// Mitsubishi GX Developer project: 20170103   PLC: FX1N

PROGRAM MAIN
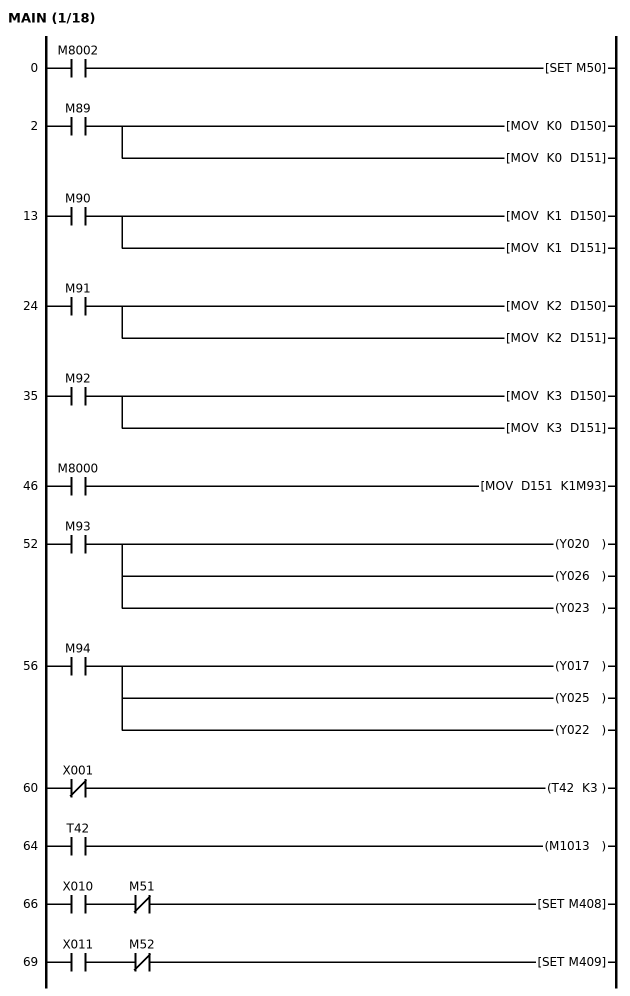
0     LD      M8002
      SET     M50
2     LD      M89
      MOV     K0 D150
      MOV     K0 D151
13    LD      M90
      MOV     K1 D150
      MOV     K1 D151
24    LD      M91
      MOV     K2 D150
      MOV     K2 D151
35    LD      M92
      MOV     K3 D150
      MOV     K3 D151
46    LD      M8000
      MOV     D151 K1M93
52    LD      M93
      OUT     Y020
      OUT     Y026
      OUT     Y023
56    LD      M94
      OUT     Y017
      OUT     Y025
      OUT     Y022
60    LDI     X001
      OUT     T42 K3
64    LD      T42
      OUT     M1013
66    LD      X010
      ANI     M51
      SET     M408
69    LD      X011
      ANI     M52
      SET     M409
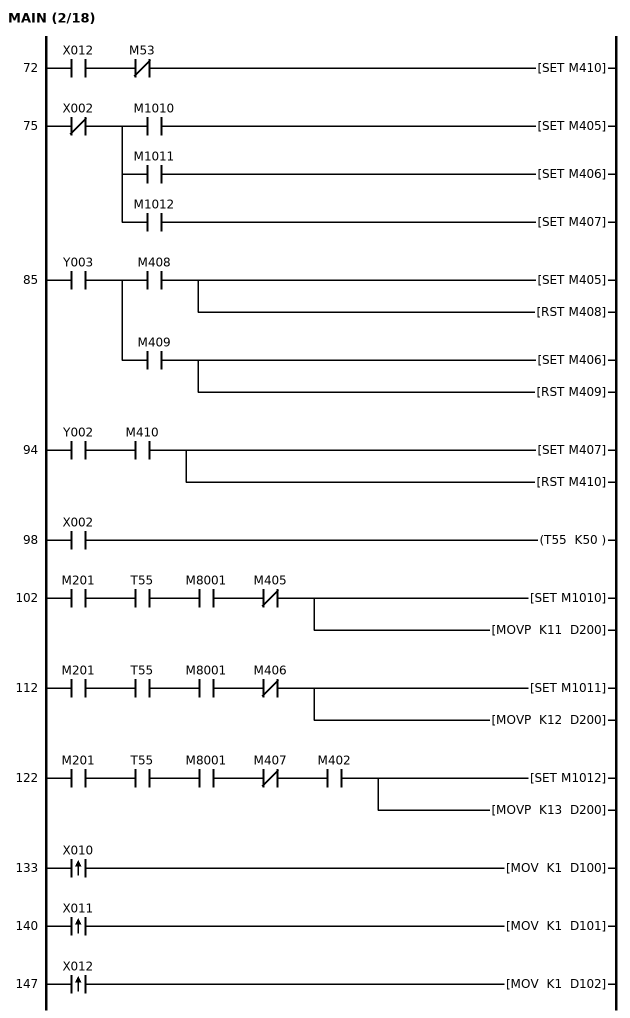
72    LD      X012
      ANI     M53
      SET     M410
75    LDI     X002
      MPS
      AND     M1010
      SET     M405
      MRD
      AND     M1011
      SET     M406
      MPP
      AND     M1012
      SET     M407
85    LD      Y003
      MPS
      AND     M408
      SET     M405
      RST     M408
      MPP
      AND     M409
      SET     M406
      RST     M409
94    LD      Y002
      AND     M410
      SET     M407
      RST     M410
98    LD      X002
      OUT     T55 K50
102   LD      M201
      AND     T55
      AND     M8001
      ANI     M405
      SET     M1010
      MOVP    K11 D200
112   LD      M201
      AND     T55
      AND     M8001
      ANI     M406
      SET     M1011
      MOVP    K12 D200
122   LD      M201
      AND     T55
      AND     M8001
      ANI     M407
      AND     M402
      SET     M1012
      MOVP    K13 D200
133   LDP     X010
      MOV     K1 D100
140   LDP     X011
      MOV     K1 D101
147   LDP     X012
      MOV     K1 D102
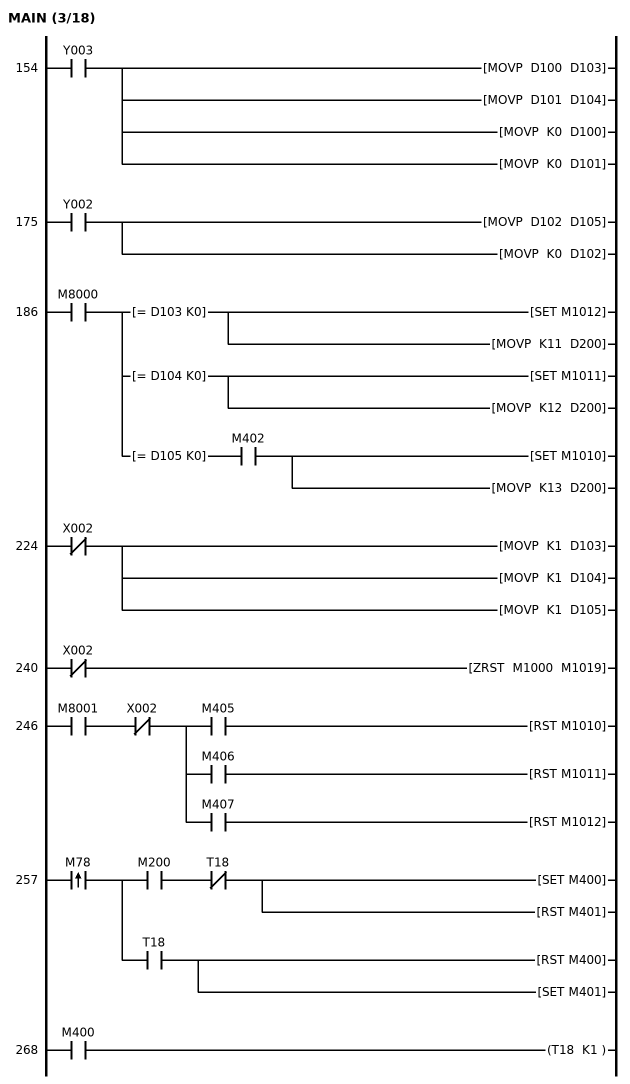
154   LD      Y003
      MOVP    D100 D103
      MOVP    D101 D104
      MOVP    K0 D100
      MOVP    K0 D101
175   LD      Y002
      MOVP    D102 D105
      MOVP    K0 D102
186   LD      M8000
      MPS
      AND=    D103 K0
      SET     M1012
      MOVP    K11 D200
      MRD
      AND=    D104 K0
      SET     M1011
      MOVP    K12 D200
      MPP
      AND=    D105 K0
      AND     M402
      SET     M1010
      MOVP    K13 D200
224   LDI     X002
      MOVP    K1 D103
      MOVP    K1 D104
      MOVP    K1 D105
240   LDI     X002
      ZRST    M1000 M1019
246   LD      M8001
      ANI     X002
      MPS
      AND     M405
      RST     M1010
      MRD
      AND     M406
      RST     M1011
      MPP
      AND     M407
      RST     M1012
257   LDP     M78
      MPS
      AND     M200
      ANI     T18
      SET     M400
      RST     M401
      MPP
      AND     T18
      RST     M400
      SET     M401
268   LD      M400
      OUT     T18 K1
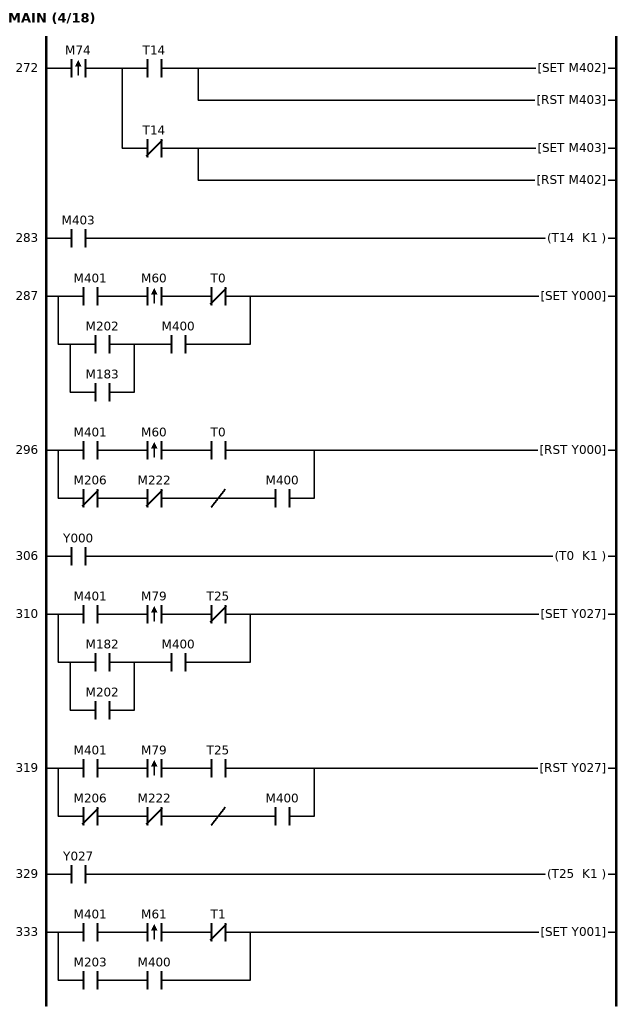
272   LDP     M74
      MPS
      AND     T14
      SET     M402
      RST     M403
      MPP
      ANI     T14
      SET     M403
      RST     M402
283   LD      M403
      OUT     T14 K1
287   LD      M401
      ANDP    M60
      ANI     T0
      LD      M202
      OR      M183
      AND     M400
      ORB
      SET     Y000
296   LD      M401
      ANDP    M60
      AND     T0
      LDI     M206
      ANI     M222
      INV
      AND     M400
      ORB
      RST     Y000
306   LD      Y000
      OUT     T0 K1
310   LD      M401
      ANDP    M79
      ANI     T25
      LD      M182
      OR      M202
      AND     M400
      ORB
      SET     Y027
319   LD      M401
      ANDP    M79
      AND     T25
      LDI     M206
      ANI     M222
      INV
      AND     M400
      ORB
      RST     Y027
329   LD      Y027
      OUT     T25 K1
333   LD      M401
      ANDP    M61
      ANI     T1
      LD      M203
      AND     M400
      ORB
      SET     Y001
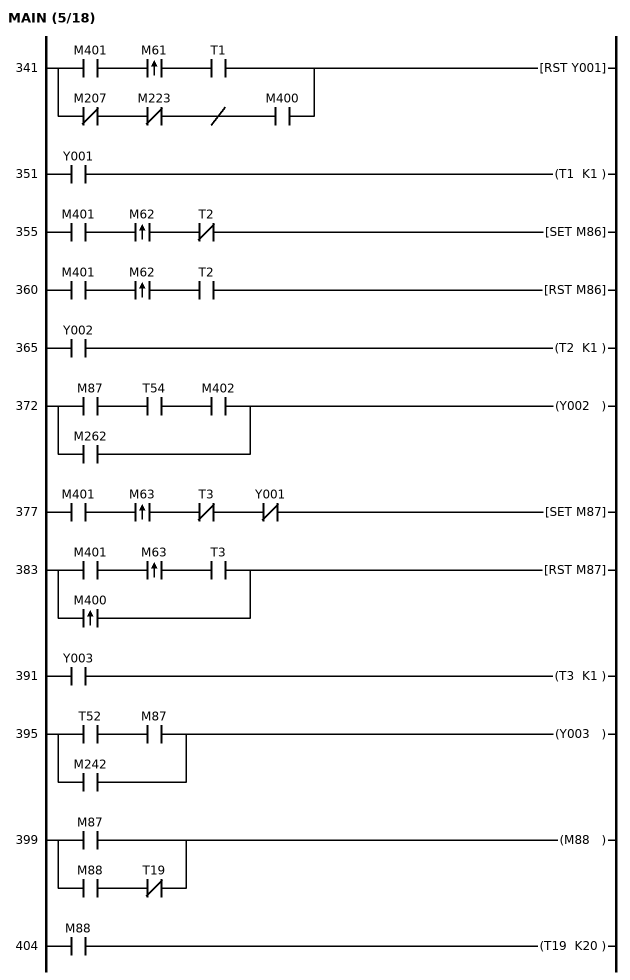
341   LD      M401
      ANDP    M61
      AND     T1
      LDI     M207
      ANI     M223
      INV
      AND     M400
      ORB
      RST     Y001
351   LD      Y001
      OUT     T1 K1
355   LD      M401
      ANDP    M62
      ANI     T2
      SET     M86
360   LD      M401
      ANDP    M62
      AND     T2
      RST     M86
365   LD      Y002
      OUT     T2 K1
372   LD      M87
      AND     T54
      AND     M402
      OR      M262
      OUT     Y002
377   LD      M401
      ANDP    M63
      ANI     T3
      ANI     Y001
      SET     M87
383   LD      M401
      ANDP    M63
      AND     T3
      ORP     M400
      RST     M87
391   LD      Y003
      OUT     T3 K1
395   LD      T52
      AND     M87
      OR      M242
      OUT     Y003
399   LD      M87
      LD      M88
      ANI     T19
      ORB
      OUT     M88
404   LD      M88
      OUT     T19 K20
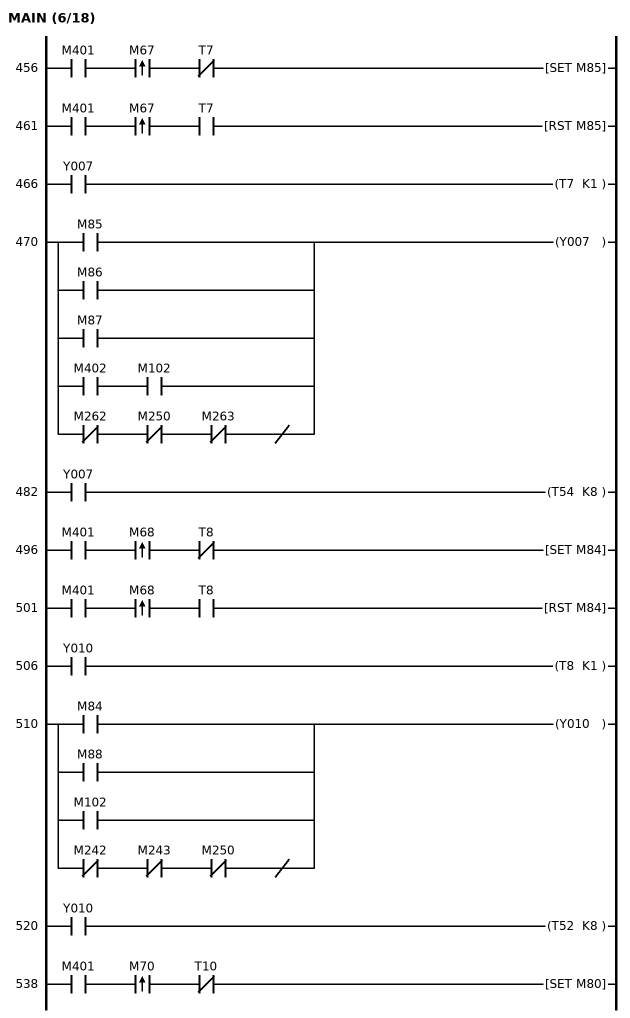
456   LD      M401
      ANDP    M67
      ANI     T7
      SET     M85
461   LD      M401
      ANDP    M67
      AND     T7
      RST     M85
466   LD      Y007
      OUT     T7 K1
470   LD      M85
      OR      M86
      OR      M87
      LD      M402
      AND     M102
      ORB
      LDI     M262
      ANI     M250
      ANI     M263
      INV
      ORB
      OUT     Y007
482   LD      Y007
      OUT     T54 K8
496   LD      M401
      ANDP    M68
      ANI     T8
      SET     M84
501   LD      M401
      ANDP    M68
      AND     T8
      RST     M84
506   LD      Y010
      OUT     T8 K1
510   LD      M84
      OR      M88
      OR      M102
      LDI     M242
      ANI     M243
      ANI     M250
      INV
      ORB
      OUT     Y010
520   LD      Y010
      OUT     T52 K8
538   LD      M401
      ANDP    M70
      ANI     T10
      SET     M80
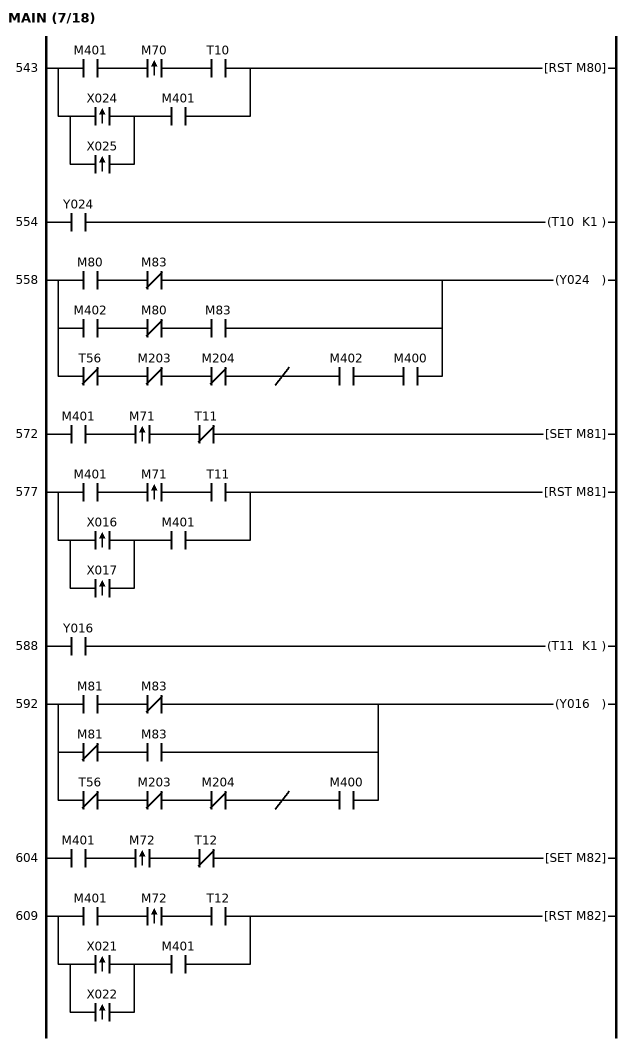
543   LD      M401
      ANDP    M70
      AND     T10
      LDP     X024
      ORP     X025
      AND     M401
      ORB
      RST     M80
554   LD      Y024
      OUT     T10 K1
558   LD      M80
      ANI     M83
      LD      M402
      ANI     M80
      AND     M83
      ORB
      LDI     T56
      ANI     M203
      ANI     M204
      INV
      AND     M402
      AND     M400
      ORB
      OUT     Y024
572   LD      M401
      ANDP    M71
      ANI     T11
      SET     M81
577   LD      M401
      ANDP    M71
      AND     T11
      LDP     X016
      ORP     X017
      AND     M401
      ORB
      RST     M81
588   LD      Y016
      OUT     T11 K1
592   LD      M81
      ANI     M83
      LDI     M81
      AND     M83
      ORB
      LDI     T56
      ANI     M203
      ANI     M204
      INV
      AND     M400
      ORB
      OUT     Y016
604   LD      M401
      ANDP    M72
      ANI     T12
      SET     M82
609   LD      M401
      ANDP    M72
      AND     T12
      LDP     X021
      ORP     X022
      AND     M401
      ORB
      RST     M82
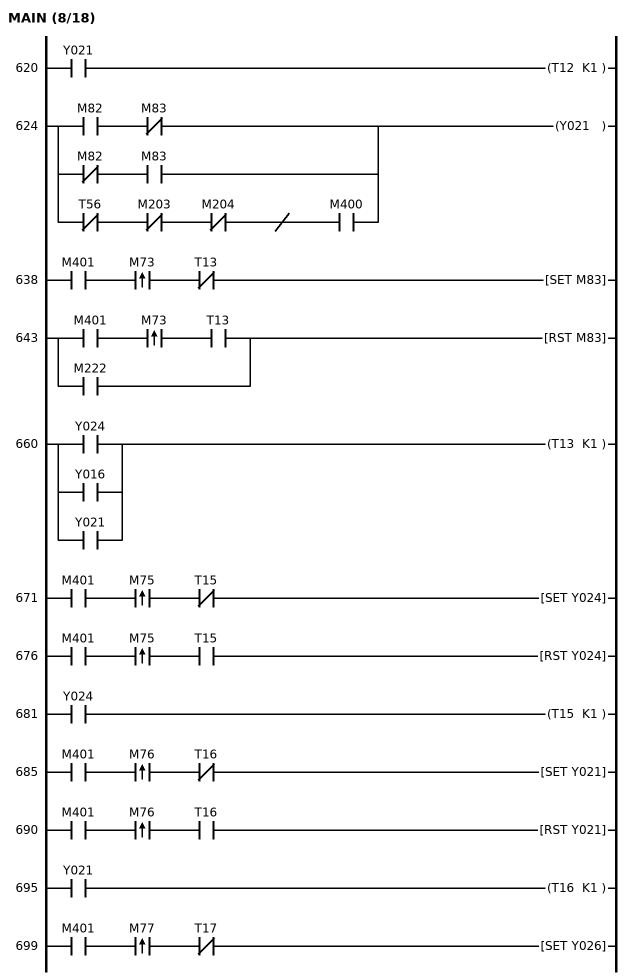
620   LD      Y021
      OUT     T12 K1
624   LD      M82
      ANI     M83
      LDI     M82
      AND     M83
      ORB
      LDI     T56
      ANI     M203
      ANI     M204
      INV
      AND     M400
      ORB
      OUT     Y021
638   LD      M401
      ANDP    M73
      ANI     T13
      SET     M83
643   LD      M401
      ANDP    M73
      AND     T13
      OR      M222
      RST     M83
660   LD      Y024
      OR      Y016
      OR      Y021
      OUT     T13 K1
671   LD      M401
      ANDP    M75
      ANI     T15
      SET     Y024
676   LD      M401
      ANDP    M75
      AND     T15
      RST     Y024
681   LD      Y024
      OUT     T15 K1
685   LD      M401
      ANDP    M76
      ANI     T16
      SET     Y021
690   LD      M401
      ANDP    M76
      AND     T16
      RST     Y021
695   LD      Y021
      OUT     T16 K1
699   LD      M401
      ANDP    M77
      ANI     T17
      SET     Y026
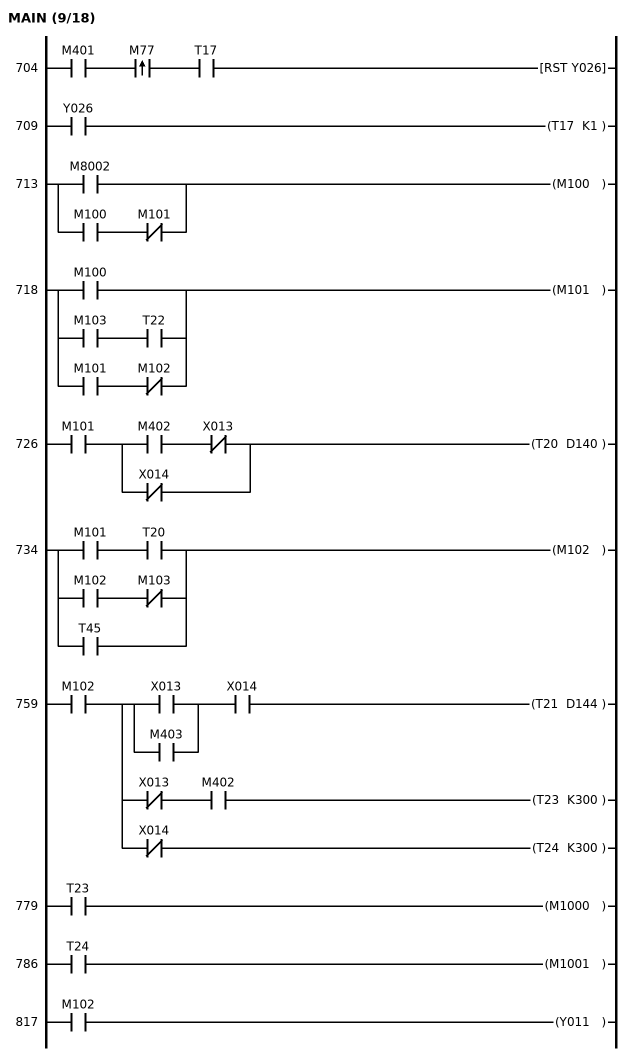
704   LD      M401
      ANDP    M77
      AND     T17
      RST     Y026
709   LD      Y026
      OUT     T17 K1
713   LD      M8002
      LD      M100
      ANI     M101
      ORB
      OUT     M100
718   LD      M100
      LD      M103
      AND     T22
      ORB
      LD      M101
      ANI     M102
      ORB
      OUT     M101
726   LD      M101
      LD      M402
      ANI     X013
      ORI     X014
      ANB
      OUT     T20 D140
734   LD      M101
      AND     T20
      LD      M102
      ANI     M103
      ORB
      OR      T45
      OUT     M102
759   LD      M102
      MPS
      LD      X013
      OR      M403
      ANB
      AND     X014
      OUT     T21 D144
      MRD
      ANI     X013
      AND     M402
      OUT     T23 K300
      MPP
      ANI     X014
      OUT     T24 K300
779   LD      T23
      OUT     M1000
786   LD      T24
      OUT     M1001
817   LD      M102
      OUT     Y011
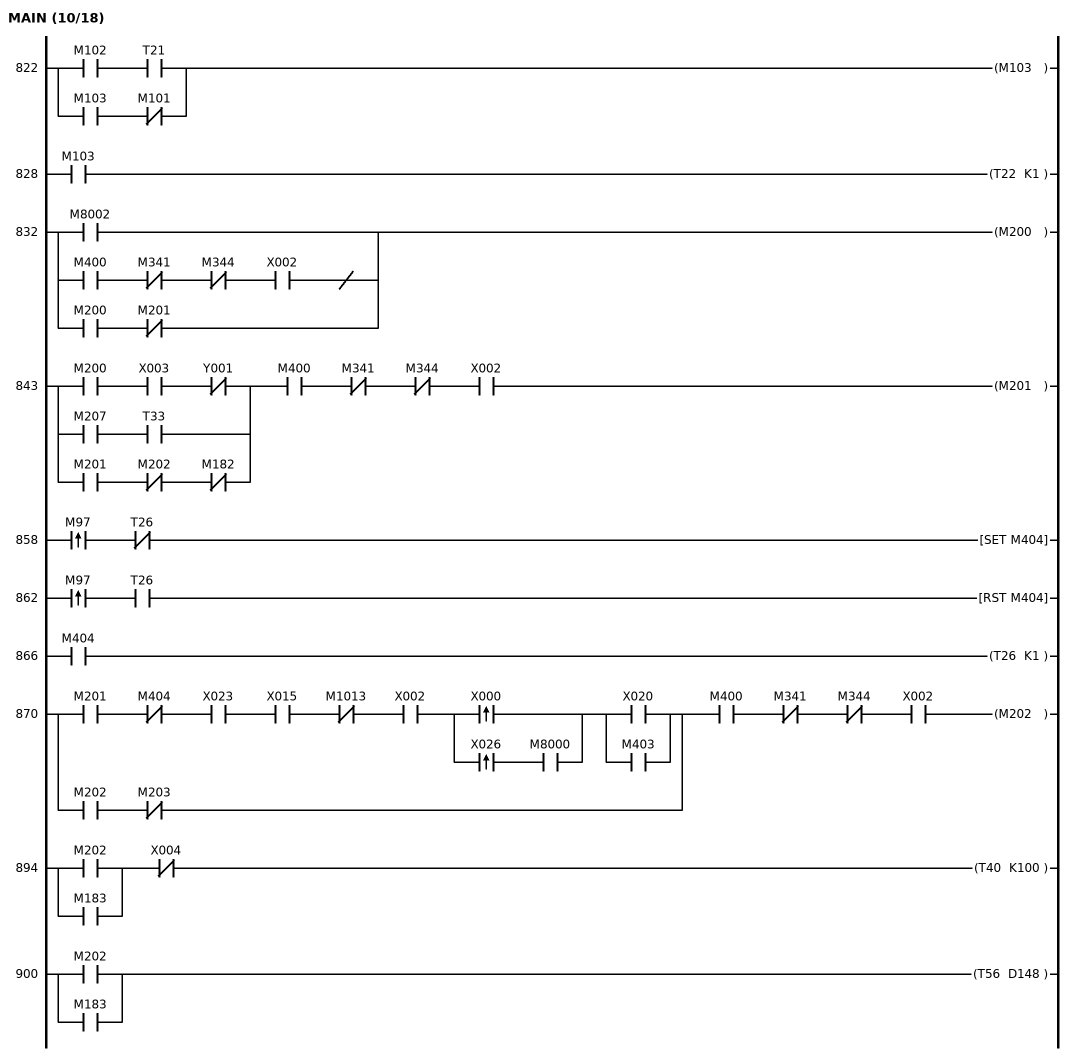
822   LD      M102
      AND     T21
      LD      M103
      ANI     M101
      ORB
      OUT     M103
828   LD      M103
      OUT     T22 K1
832   LD      M8002
      LD      M400
      ANI     M341
      ANI     M344
      AND     X002
      INV
      ORB
      LD      M200
      ANI     M201
      ORB
      OUT     M200
843   LD      M200
      AND     X003
      ANI     Y001
      LD      M207
      AND     T33
      ORB
      LD      M201
      ANI     M202
      ANI     M182
      ORB
      AND     M400
      ANI     M341
      ANI     M344
      AND     X002
      OUT     M201
858   LDP     M97
      ANI     T26
      SET     M404
862   LDP     M97
      AND     T26
      RST     M404
866   LD      M404
      OUT     T26 K1
870   LD      M201
      ANI     M404
      AND     X023
      AND     X015
      ANI     M1013
      AND     X002
      LDP     X000
      LDP     X026
      AND     M8000
      ORB
      ANB
      LD      X020
      OR      M403
      ANB
      LD      M202
      ANI     M203
      ORB
      AND     M400
      ANI     M341
      ANI     M344
      AND     X002
      OUT     M202
894   LD      M202
      OR      M183
      ANI     X004
      OUT     T40 K100
900   LD      M202
      OR      M183
      OUT     T56 D148
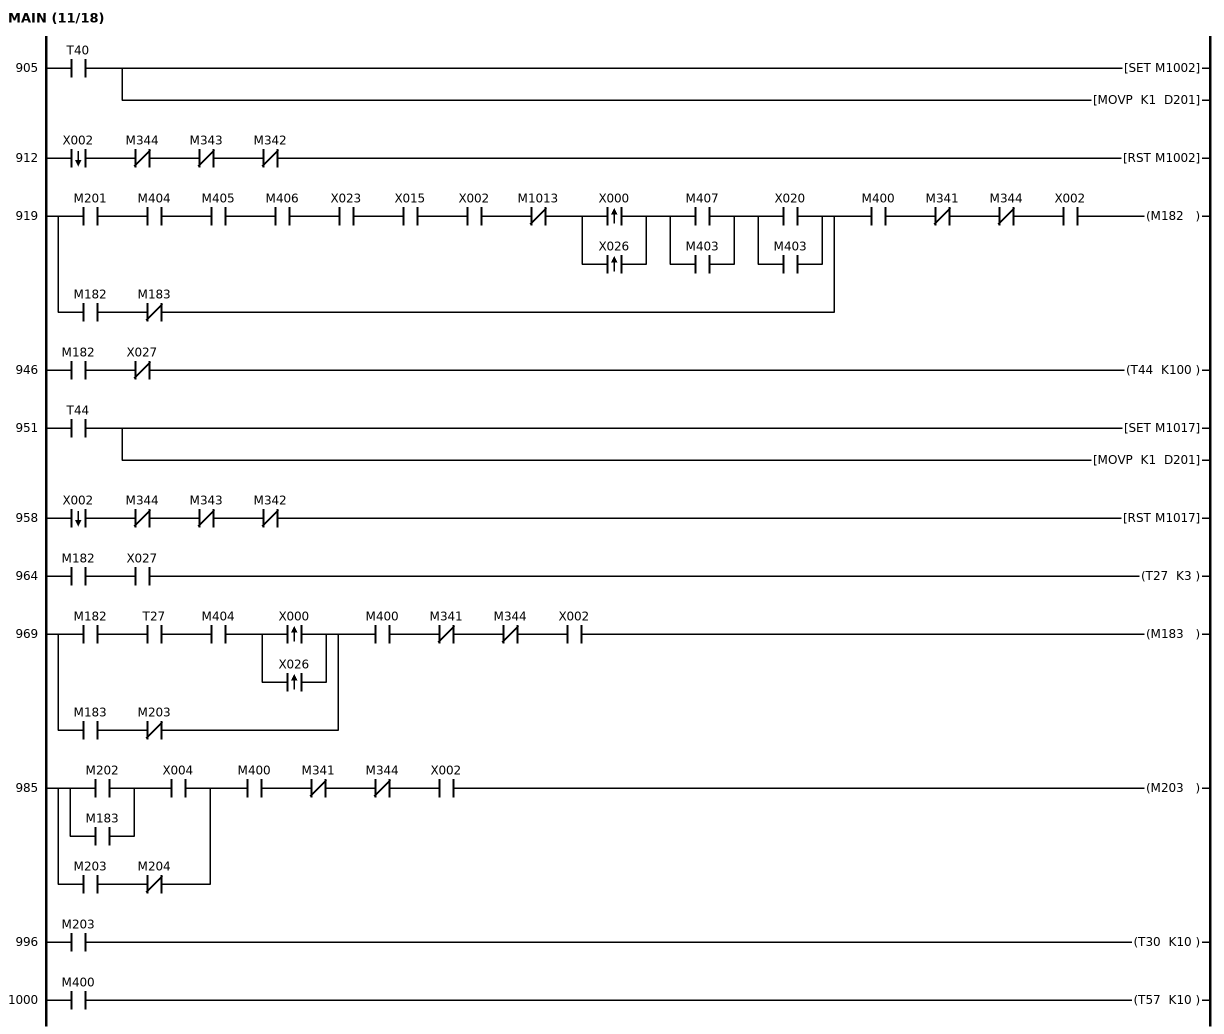
905   LD      T40
      SET     M1002
      MOVP    K1 D201
912   LDF     X002
      ANI     M344
      ANI     M343
      ANI     M342
      RST     M1002
919   LD      M201
      AND     M404
      AND     M405
      AND     M406
      AND     X023
      AND     X015
      AND     X002
      ANI     M1013
      LDP     X000
      ORP     X026
      ANB
      LD      M407
      OR      M403
      ANB
      LD      X020
      OR      M403
      ANB
      LD      M182
      ANI     M183
      ORB
      AND     M400
      ANI     M341
      ANI     M344
      AND     X002
      OUT     M182
946   LD      M182
      ANI     X027
      OUT     T44 K100
951   LD      T44
      SET     M1017
      MOVP    K1 D201
958   LDF     X002
      ANI     M344
      ANI     M343
      ANI     M342
      RST     M1017
964   LD      M182
      AND     X027
      OUT     T27 K3
969   LD      M182
      AND     T27
      AND     M404
      LDP     X000
      ORP     X026
      ANB
      LD      M183
      ANI     M203
      ORB
      AND     M400
      ANI     M341
      ANI     M344
      AND     X002
      OUT     M183
985   LD      M202
      OR      M183
      AND     X004
      LD      M203
      ANI     M204
      ORB
      AND     M400
      ANI     M341
      ANI     M344
      AND     X002
      OUT     M203
996   LD      M203
      OUT     T30 K10
1000  LD      M400
      OUT     T57 K10
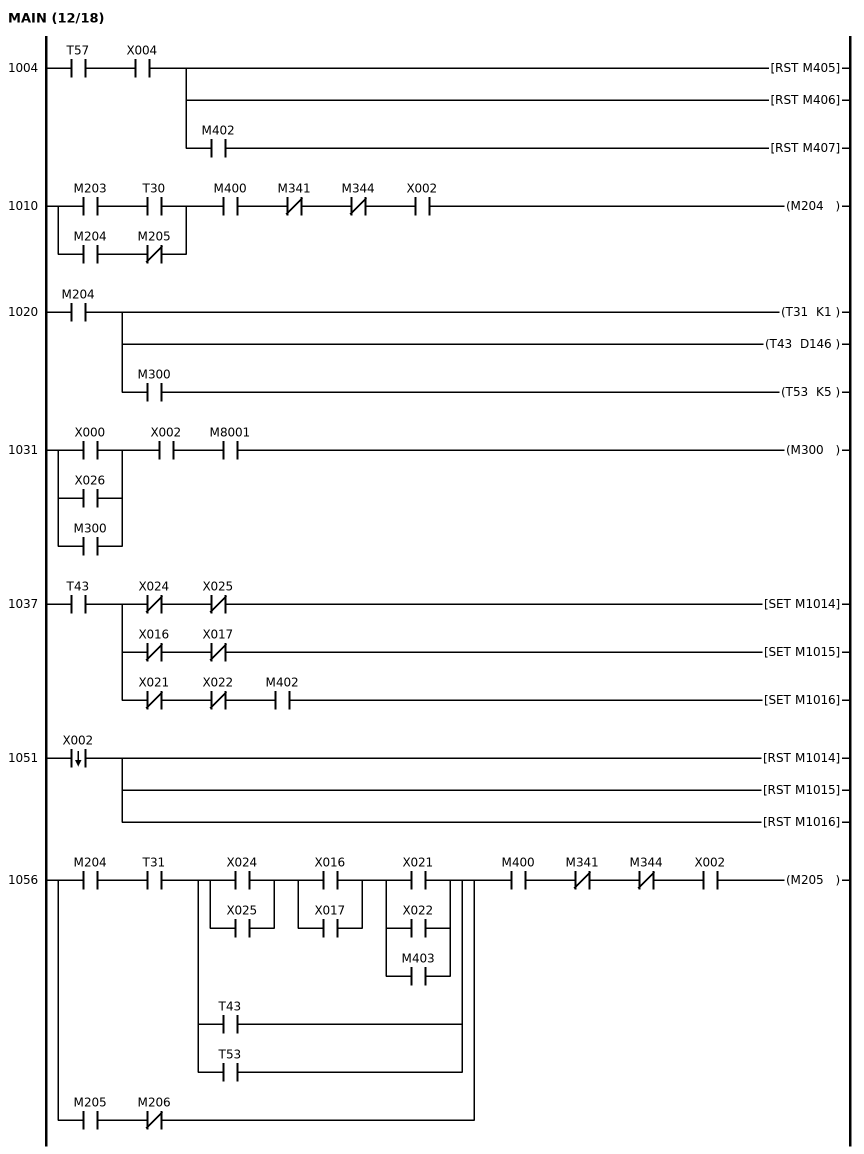
1004  LD      T57
      AND     X004
      RST     M405
      RST     M406
      AND     M402
      RST     M407
1010  LD      M203
      AND     T30
      LD      M204
      ANI     M205
      ORB
      AND     M400
      ANI     M341
      ANI     M344
      AND     X002
      OUT     M204
1020  LD      M204
      OUT     T31 K1
      OUT     T43 D146
      AND     M300
      OUT     T53 K5
1031  LD      X000
      OR      X026
      OR      M300
      AND     X002
      AND     M8001
      OUT     M300
1037  LD      T43
      MPS
      ANI     X024
      ANI     X025
      SET     M1014
      MRD
      ANI     X016
      ANI     X017
      SET     M1015
      MPP
      ANI     X021
      ANI     X022
      AND     M402
      SET     M1016
1051  LDF     X002
      RST     M1014
      RST     M1015
      RST     M1016
1056  LD      M204
      AND     T31
      LD      X024
      OR      X025
      LD      X016
      OR      X017
      ANB
      LD      X021
      OR      X022
      OR      M403
      ANB
      OR      T43
      OR      T53
      ANB
      LD      M205
      ANI     M206
      ORB
      AND     M400
      ANI     M341
      ANI     M344
      AND     X002
      OUT     M205
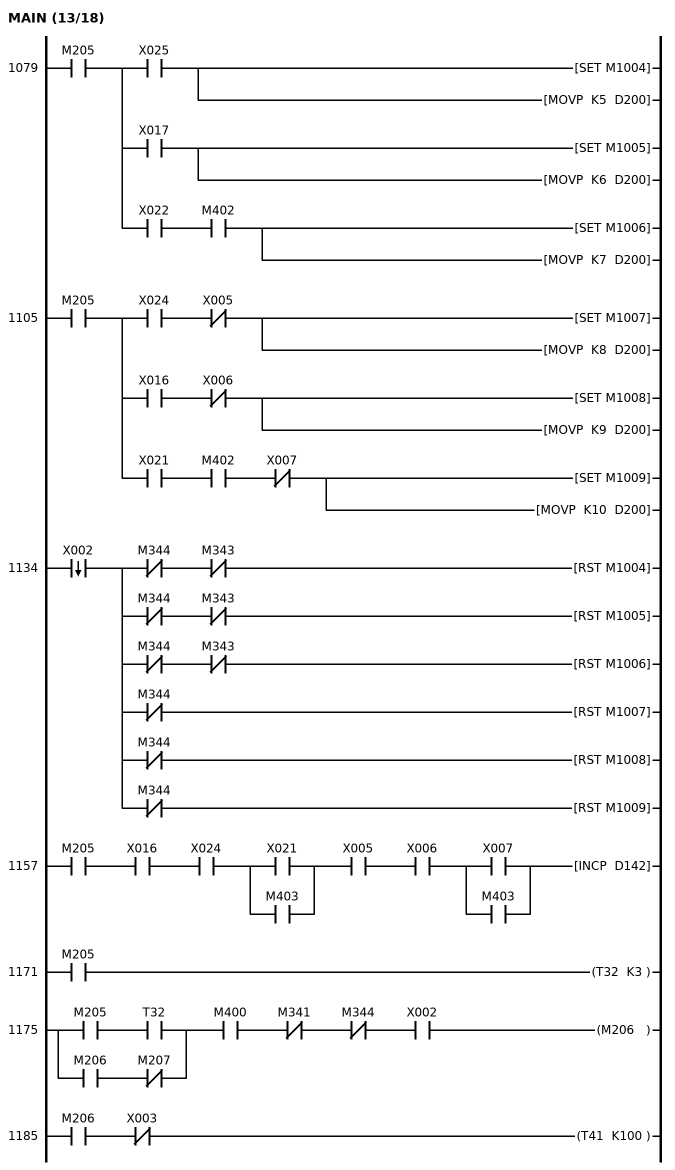
1079  LD      M205
      MPS
      AND     X025
      SET     M1004
      MOVP    K5 D200
      MRD
      AND     X017
      SET     M1005
      MOVP    K6 D200
      MPP
      AND     X022
      AND     M402
      SET     M1006
      MOVP    K7 D200
1105  LD      M205
      MPS
      AND     X024
      ANI     X005
      SET     M1007
      MOVP    K8 D200
      MRD
      AND     X016
      ANI     X006
      SET     M1008
      MOVP    K9 D200
      MPP
      AND     X021
      AND     M402
      ANI     X007
      SET     M1009
      MOVP    K10 D200
1134  LDF     X002
      MPS
      ANI     M344
      ANI     M343
      RST     M1004
      MRD
      ANI     M344
      ANI     M343
      RST     M1005
      MRD
      ANI     M344
      ANI     M343
      RST     M1006
      MRD
      ANI     M344
      RST     M1007
      MRD
      ANI     M344
      RST     M1008
      MPP
      ANI     M344
      RST     M1009
1157  LD      M205
      AND     X016
      AND     X024
      LD      X021
      OR      M403
      ANB
      AND     X005
      AND     X006
      LD      X007
      OR      M403
      ANB
      INCP    D142
1171  LD      M205
      OUT     T32 K3
1175  LD      M205
      AND     T32
      LD      M206
      ANI     M207
      ORB
      AND     M400
      ANI     M341
      ANI     M344
      AND     X002
      OUT     M206
1185  LD      M206
      ANI     X003
      OUT     T41 K100
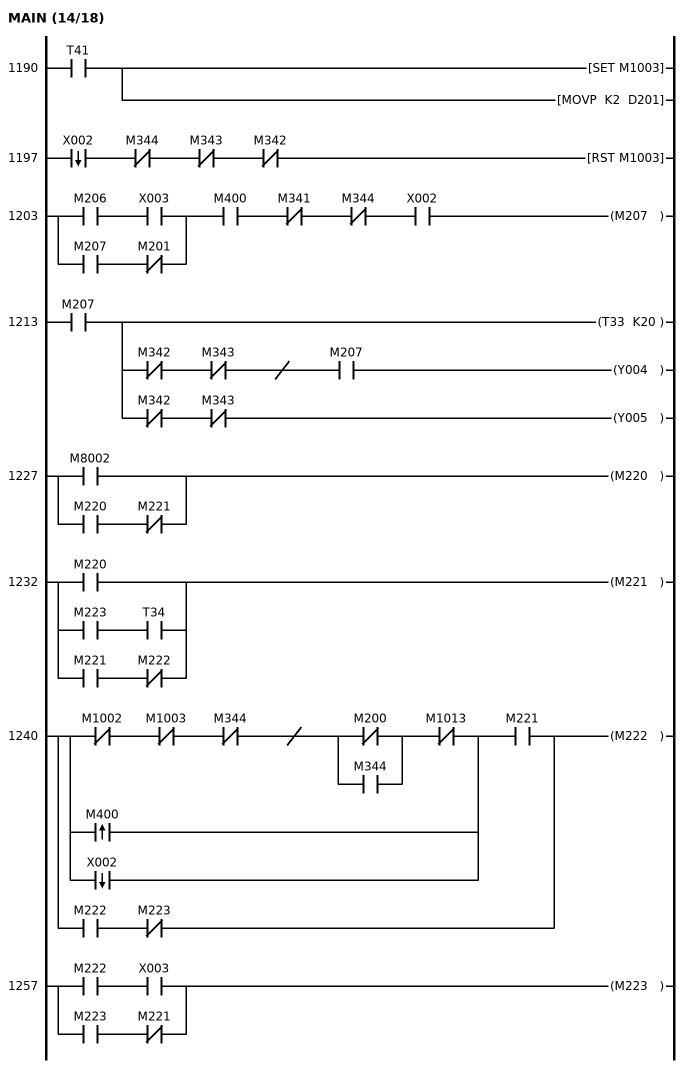
1190  LD      T41
      SET     M1003
      MOVP    K2 D201
1197  LDF     X002
      ANI     M344
      ANI     M343
      ANI     M342
      RST     M1003
1203  LD      M206
      AND     X003
      LD      M207
      ANI     M201
      ORB
      AND     M400
      ANI     M341
      ANI     M344
      AND     X002
      OUT     M207
1213  LD      M207
      OUT     T33 K20
      MPS
      ANI     M342
      ANI     M343
      INV
      AND     M207
      OUT     Y004
      MPP
      ANI     M342
      ANI     M343
      OUT     Y005
1227  LD      M8002
      LD      M220
      ANI     M221
      ORB
      OUT     M220
1232  LD      M220
      LD      M223
      AND     T34
      ORB
      LD      M221
      ANI     M222
      ORB
      OUT     M221
1240  LDI     M1002
      ANI     M1003
      ANI     M344
      INV
      LDI     M200
      OR      M344
      ANB
      ANI     M1013
      ORP     M400
      ORF     X002
      AND     M221
      LD      M222
      ANI     M223
      ORB
      OUT     M222
1257  LD      M222
      AND     X003
      LD      M223
      ANI     M221
      ORB
      OUT     M223
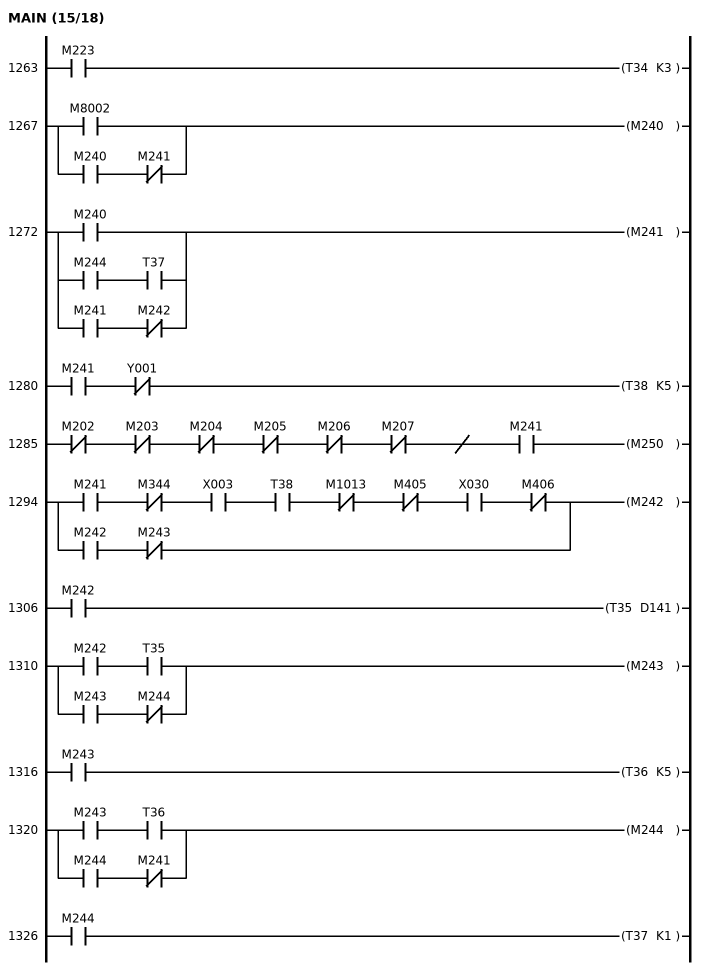
1263  LD      M223
      OUT     T34 K3
1267  LD      M8002
      LD      M240
      ANI     M241
      ORB
      OUT     M240
1272  LD      M240
      LD      M244
      AND     T37
      ORB
      LD      M241
      ANI     M242
      ORB
      OUT     M241
1280  LD      M241
      ANI     Y001
      OUT     T38 K5
1285  LDI     M202
      ANI     M203
      ANI     M204
      ANI     M205
      ANI     M206
      ANI     M207
      INV
      AND     M241
      OUT     M250
1294  LD      M241
      ANI     M344
      AND     X003
      AND     T38
      ANI     M1013
      ANI     M405
      AND     X030
      ANI     M406
      LD      M242
      ANI     M243
      ORB
      OUT     M242
1306  LD      M242
      OUT     T35 D141
1310  LD      M242
      AND     T35
      LD      M243
      ANI     M244
      ORB
      OUT     M243
1316  LD      M243
      OUT     T36 K5
1320  LD      M243
      AND     T36
      LD      M244
      ANI     M241
      ORB
      OUT     M244
1326  LD      M244
      OUT     T37 K1
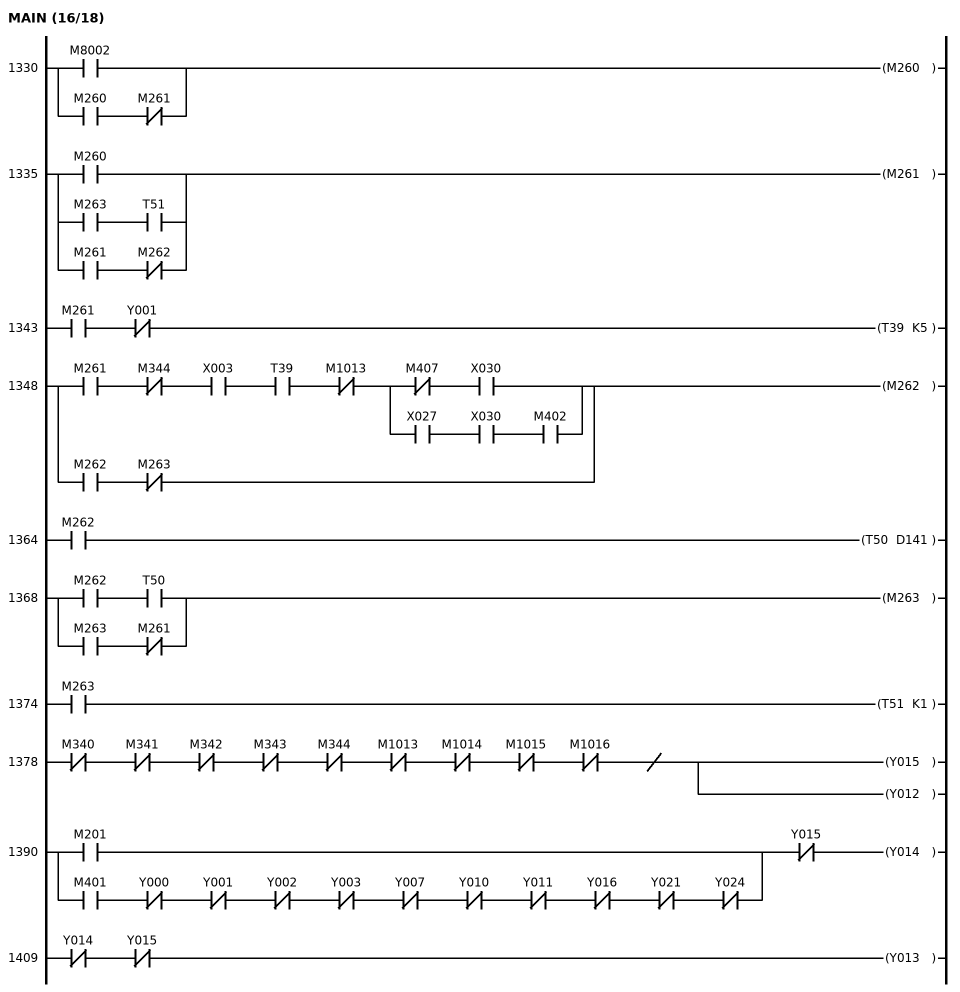
1330  LD      M8002
      LD      M260
      ANI     M261
      ORB
      OUT     M260
1335  LD      M260
      LD      M263
      AND     T51
      ORB
      LD      M261
      ANI     M262
      ORB
      OUT     M261
1343  LD      M261
      ANI     Y001
      OUT     T39 K5
1348  LD      M261
      ANI     M344
      AND     X003
      AND     T39
      ANI     M1013
      LDI     M407
      AND     X030
      LD      X027
      AND     X030
      AND     M402
      ORB
      ANB
      LD      M262
      ANI     M263
      ORB
      OUT     M262
1364  LD      M262
      OUT     T50 D141
1368  LD      M262
      AND     T50
      LD      M263
      ANI     M261
      ORB
      OUT     M263
1374  LD      M263
      OUT     T51 K1
1378  LDI     M340
      ANI     M341
      ANI     M342
      ANI     M343
      ANI     M344
      ANI     M1013
      ANI     M1014
      ANI     M1015
      ANI     M1016
      INV
      OUT     Y015
      OUT     Y012
1390  LD      M201
      LD      M401
      ANI     Y000
      ANI     Y001
      ANI     Y002
      ANI     Y003
      ANI     Y007
      ANI     Y010
      ANI     Y011
      ANI     Y016
      ANI     Y021
      ANI     Y024
      ORB
      ANI     Y015
      OUT     Y014
1409  LDI     Y014
      ANI     Y015
      OUT     Y013
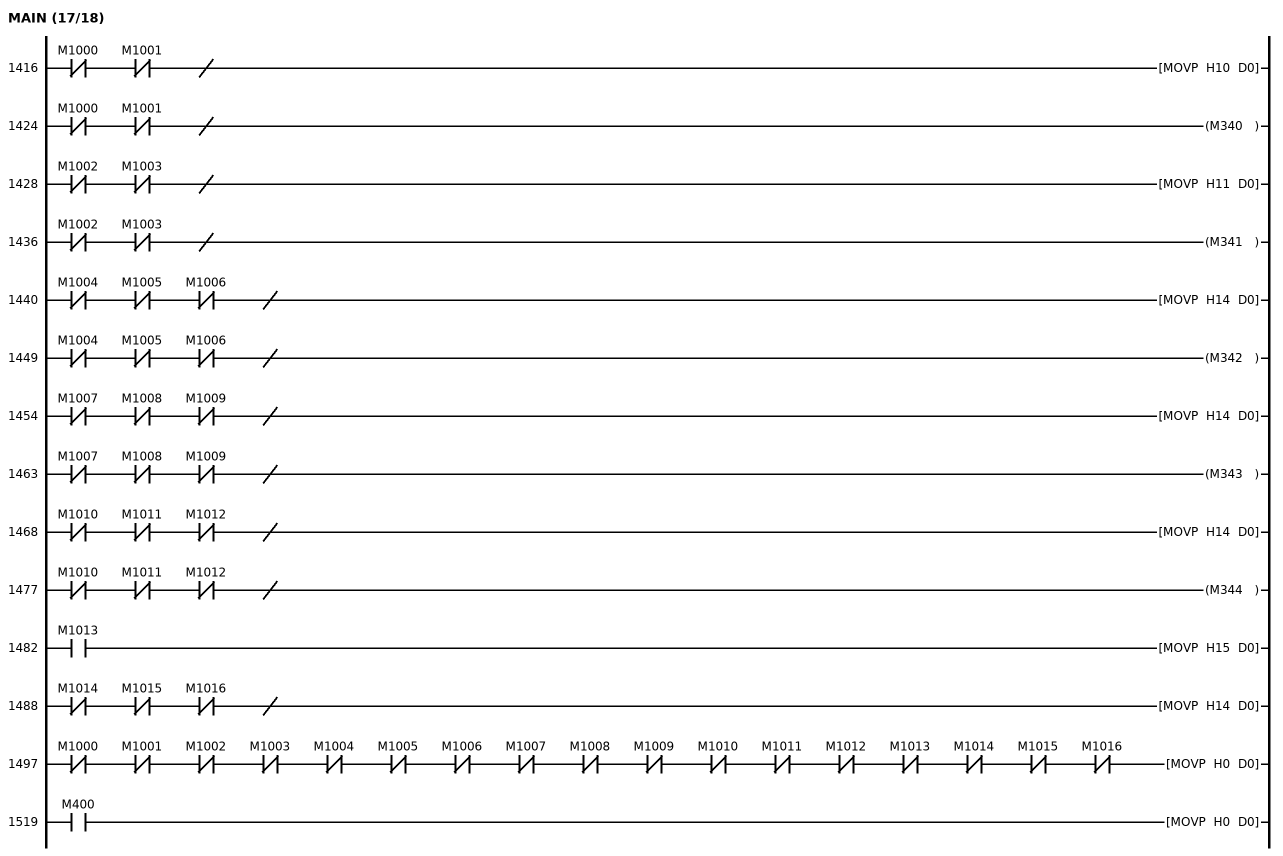
1416  LDI     M1000
      ANI     M1001
      INV
      MOVP    H10 D0
1424  LDI     M1000
      ANI     M1001
      INV
      OUT     M340
1428  LDI     M1002
      ANI     M1003
      INV
      MOVP    H11 D0
1436  LDI     M1002
      ANI     M1003
      INV
      OUT     M341
1440  LDI     M1004
      ANI     M1005
      ANI     M1006
      INV
      MOVP    H14 D0
1449  LDI     M1004
      ANI     M1005
      ANI     M1006
      INV
      OUT     M342
1454  LDI     M1007
      ANI     M1008
      ANI     M1009
      INV
      MOVP    H14 D0
1463  LDI     M1007
      ANI     M1008
      ANI     M1009
      INV
      OUT     M343
1468  LDI     M1010
      ANI     M1011
      ANI     M1012
      INV
      MOVP    H14 D0
1477  LDI     M1010
      ANI     M1011
      ANI     M1012
      INV
      OUT     M344
1482  LD      M1013
      MOVP    H15 D0
1488  LDI     M1014
      ANI     M1015
      ANI     M1016
      INV
      MOVP    H14 D0
1497  LDI     M1000
      ANI     M1001
      ANI     M1002
      ANI     M1003
      ANI     M1004
      ANI     M1005
      ANI     M1006
      ANI     M1007
      ANI     M1008
      ANI     M1009
      ANI     M1010
      ANI     M1011
      ANI     M1012
      ANI     M1013
      ANI     M1014
      ANI     M1015
      ANI     M1016
      MOVP    H0 D0
1519  LD      M400
      MOVP    H0 D0
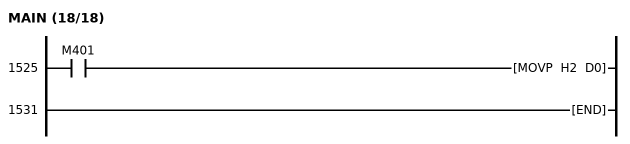
1525  LD      M401
      MOVP    H2 D0
1531  END
END_PROGRAM
